FUNCTION F_GetValvePosition : SINT
VAR_INPUT
	iValveIndex	: USINT; // Valve index
END_VAR
VAR
	rValveActualPos		: LREAL; // valve actual position
	rPositionTolerance	: REAL := 2.0;
END_VAR

//Funtion to get the actual valve position
rValveActualPos := GVL_Motion.aValves[iValveIndex].rActualPos;

IF rValveActualPos > 0 - rPositionTolerance AND rValveActualPos < 0 + rPositionTolerance THEN
	F_GetValvePosition := 1;
	RETURN;
END_IF

IF rValveActualPos > 1200 - rPositionTolerance AND rValveActualPos < 1200 + rPositionTolerance THEN
	F_GetValvePosition := 2;
	RETURN;
END_IF

IF rValveActualPos > 2400 - rPositionTolerance AND rValveActualPos < 2400 + rPositionTolerance THEN
	F_GetValvePosition := 3;
	RETURN;
END_IF

IF rValveActualPos > 3600 - rPositionTolerance AND rValveActualPos < 3600 + rPositionTolerance THEN
	F_GetValvePosition := 4;
	RETURN;
END_IF

IF rValveActualPos > 4800 - rPositionTolerance AND rValveActualPos < 4800 + rPositionTolerance THEN
	F_GetValvePosition := 5;
	RETURN;
END_IF

IF rValveActualPos > 6000 - rPositionTolerance AND rValveActualPos < 6000 + rPositionTolerance THEN
	F_GetValvePosition := 6;
	RETURN;
END_IF

F_GetValvePosition := -1;
RETURN;

END_FUNCTION

(* stored: Version 1.1.0.1, ProductVersion 3.1.4024.12
   POU F_GetValvePosition: Id {ecae4da1-5a18-4e05-8b47-a24f0fbafec2}, SpecialFunc None *)
